// TwinCAT 3 PLC project Project
// ProgramVersion: 3.1.4023.0
// libraries:
//   Tc2_EtherCAT, * (Beckhoff Automation GmbH)
//   Tc2_Standard, * (Beckhoff Automation GmbH)
//   Tc2_System, * (Beckhoff Automation GmbH)
//   Tc2_Utilities, * (Beckhoff Automation GmbH)
//   Tc3_Module, * (Beckhoff Automation GmbH)
// project tree:
//   DUTs/ EtherCATDiagnosisState.TcDUT, SlaveInfo.TcDUT
//   GVLs/ GVL.TcGVL
//   / PlcTask.TcTTO
//   POUs/EtherCAT Monitoring/ FB_Diag_ECAT_Module.TcPOU, FB_EtherCATInit.TcPOU, FB_ReadSlavesEherCAT.TcPOU, SIC_Diagnosis_Modules.TcPOU
//   POUs/ MAIN.TcPOU
// real-time tasks:
//   TASK PlcTask: cycle T#1ms, priority 20, ADS port 350
// I/O:
//   DEVICE Device 1 (EtherCAT), AmsNetId 192.168.212.233.2.1
//     SyncCRIO (NI 9145) [NI 9145]
//     AZ5 (TW.LSST.AZIMUTH) [TW.LSST.AZIMUTH]
//     AZ6 (TW.LSST.AZIMUTH) [TW.LSST.AZIMUTH]
//     AZ7 (TW.LSST.AZIMUTH) [TW.LSST.AZIMUTH]
//     AZ8 (TW.LSST.AZIMUTH) [TW.LSST.AZIMUTH]
//     AZ_HS (LSST.HS.board) [LSST.HS.board]
//     AZ16 (TW.LSST.AZIMUTH) [TW.LSST.AZIMUTH]
//     AZ15 (TW.LSST.AZIMUTH) [TW.LSST.AZIMUTH]
//     AZ14 (TW.LSST.AZIMUTH) [TW.LSST.AZIMUTH]
//     AZ13 (TW.LSST.AZIMUTH) [TW.LSST.AZIMUTH]
//     EL51 (TW.LSST.ALTITUDE) [TW.LSST.ALTITUDE]
//     EL52 (TW.LSST.ALTITUDE) [TW.LSST.ALTITUDE]
//     EL41 (TW.LSST.ALTITUDE) [TW.LSST.ALTITUDE]
//     EL42 (TW.LSST.ALTITUDE) [TW.LSST.ALTITUDE]
//     EL_XNeg_HS (LSST.HS.board) [LSST.HS.board]
//     EL61 (TW.LSST.ALTITUDE) [TW.LSST.ALTITUDE]
//     EL62 (TW.LSST.ALTITUDE) [TW.LSST.ALTITUDE]
//     AZ9 (TW.LSST.AZIMUTH) [TW.LSST.AZIMUTH]
//     AZ10 (TW.LSST.AZIMUTH) [TW.LSST.AZIMUTH]
//     AZ11 (TW.LSST.AZIMUTH) [TW.LSST.AZIMUTH]
//     AZ12 (TW.LSST.AZIMUTH) [TW.LSST.AZIMUTH]
//     AZ4 (TW.LSST.AZIMUTH) [TW.LSST.AZIMUTH]
//     AZ3 (TW.LSST.AZIMUTH) [TW.LSST.AZIMUTH]
//     AZ2 (TW.LSST.AZIMUTH) [TW.LSST.AZIMUTH]
//     AZ1 (TW.LSST.AZIMUTH) [TW.LSST.AZIMUTH] (disabled)
//     EL21 (TW.LSST.ALTITUDE) [TW.LSST.ALTITUDE]
//     EL22 (TW.LSST.ALTITUDE) [TW.LSST.ALTITUDE]
//     EL11 (TW.LSST.ALTITUDE) [TW.LSST.ALTITUDE]
//     EL12 (TW.LSST.ALTITUDE) [TW.LSST.ALTITUDE]
//     EL_XPos_HS (LSST.HS.board) [LSST.HS.board]
//     EL31 (TW.LSST.ALTITUDE) [TW.LSST.ALTITUDE]
//     EL32 (TW.LSST.ALTITUDE) [TW.LSST.ALTITUDE]
// variable links:
//   Project/Project Instance <-> Device 1 (EtherCAT)/AZ5 (TW.LSST.AZIMUTH)
//     PlcTask Inputs/MAIN.StatusWordDrive2 <-> Inputs/Status word

CONFIGURATION Project
    RESOURCE PLC ON TwinCAT3
        TASK PlcTask(INTERVAL := T#1ms, PRIORITY := 20);
        PROGRAM MAIN WITH PlcTask : MAIN;
    END_RESOURCE
END_CONFIGURATION

// ---- DUTs/EtherCATDiagnosisState.TcDUT
{attribute 'qualified_only'}
{attribute 'strict'}
TYPE EtherCATDiagnosisState :
(
	Init								:= 0,
	GetPLCAdress						:= 1,
	GetSlavesAddresses 					:= 2,
	GetSlavesConfiguration 				:= 3,
	ReadSlavesIdentity					:= 4,
	
	ReadSlaveCyclicData					:= 10,
	
	ProcessSlavesCyclicData				:= 100
);
END_TYPE

// ---- DUTs/SlaveInfo.TcDUT
TYPE SlaveInfo :
STRUCT
	Address 						: WORD;
	Name 							: STRING[31];
	ConfiguredVendorID				: UDINT;
	ConfiguredProductCode 			: UDINT;
	ConfiguredRevisionNo 			: UDINT;
	ConfiguredSerialNo				: UDINT;
	ReadVendorID					: UDINT;
	ReadProductCode 				: UDINT;
	ReadRevisionNo 					: UDINT;
	ReadSerialNo					: UDINT;
	CRCerrorCounter					: DWORD;
	stCrcError						: ST_EcCrcErrorEx;
	StateChanges					: UDINT;
	StateChangesTimes				: ARRAY [0..255] OF TIMESTRUCT;
	StateChangesIndex				: UINT;
	AbnormalStateChanges			: UDINT;
	AbnormalStateChangesTimes		: ARRAY [0..255] OF TIMESTRUCT;
	AbnormalStateChangesIndex		: UINT;
	
	
END_STRUCT
END_TYPE

// ---- GVLs/GVL.TcGVL

VAR_GLOBAL
	PLCEtherCatAddress : T_AmsNetId;
END_VAR

// ---- POUs/MAIN.TcPOU
PROGRAM MAIN
VAR
	MyVar AT%I*:UDINT;
	StatusWordDrive2 AT%I*:UINT;
	
	
	b_PLCInitialization			: BOOL;
	b_EtherCATMasterErrorRun	: BOOL;
	
	//fbEtherCatInit 			: FB_EtherCATInit;
	
	
	
	fbGetLocalAmsNetId		: FB_GetLocalAmsNetId;
	sPlcNetId				: T_AmsNetId := '192.168.212.233.1.1';
	sEcatMaterNetId       	: T_AmsNetId := '192.168.212.233.2.1';
//	fbGetEcMasterState 		: FB_EcGetMasterState;
	 fbGetAllEcSlaveStates 	: FB_EcGetAllSlaveStates;
	 
    bExecute            : BOOL := TRUE;
    devStates           : ARRAY[0..EC_MAX_SLAVES] OF ST_EcSlaveState;
    nSlaves             : UINT := 0;
    bError              : BOOL;
    nErrId              : UDINT;
	
	bFirstCall 					: BOOL := TRUE;
	fbGetAllEcSlaveAddr 		: FB_EcGetAllSlaveAddr;
	slaveAddresses    			: ARRAY[0..EC_MAX_SLAVES] OF UINT;    
    bErrorSlaveAddr           	: BOOL;
  
	
	i : UINT;
	
	fbGetSlaveIdentity : FB_EcGetSlaveIdentity;  
    identity           : ARRAY [0..EC_MAX_SLAVES] OF ST_EcSlaveIdentity;
	
	fbEcGetConfSlaves : FB_EcGetConfSlaves;
	ArrEcConfSlaveInfo : ARRAY[0..EC_MAX_SLAVES] OF ST_EcSlaveConfigData; 
	
	
	fbEcGetAllSlavesStateChanges 	: FB_EcGetAllSlavePresentStateChanges;
	ArrSlaveStateChangeBuff	  		:  ARRAY [0..EC_MAX_SLAVES] OF UDINT;
	
	fbEcGetAllSlavesCrcErrors			: FB_EcGetAllSlaveCrcErrors;
	ArrSlavesCrcErrorCounterBuff	: ARRAY [0..EC_MAX_SLAVES] OF DWORD;
	
	fbEcGetSlaveCrcError		: FB_EcGetSlaveCrcError;
	
	fbEcGetAllSlaveAbnormalStateChanges	: FB_EcGetAllSlaveAbnormalStateChanges;
	ArrSlavesAbnormalStateChanges		:  ARRAY [0..EC_MAX_SLAVES] OF UDINT; 
    
	fbGetTime : NT_GetTime;
	
   bBusy : BOOL;
   
   
   arrSlaveData : ARRAY [0..EC_MAX_SLAVES] OF SlaveInfo;

	
	lastStateChangeValue: UDINT;
	
	eDiagnosisState : EtherCATDiagnosisState := EtherCATDiagnosisState.Init;
	
END_VAR

VAR CONSTANT
	EC_MAX_SLAVES : UINT :=255;
END_VAR


CASE eDiagnosisState OF
	//Init the diagnosis
	EtherCATDiagnosisState.Init:
		bExecute := TRUE;
		eDiagnosisState := EtherCATDiagnosisState.GetPLCAdress;
		FOR i:= 0 TO EC_MAX_SLAVES DO
			arrSlaveData[i].StateChangesIndex 			:= 0;
			arrSlaveData[i].AbnormalStateChangesIndex 	:= 0;
		END_FOR
 				
	//Get PLC address
	EtherCATDiagnosisState.GetPLCAdress:
		fbGetLocalAmsNetId(bExecute:= bExecute);
		bBusy := fbGetLocalAmsNetId.bBusy;
		bError := fbGetLocalAmsNetId.bError;
		IF NOT bBusy AND NOT bError AND bExecute THEN
			sPlcNetId := fbGetLocalAmsNetId.AddrString;
			eDiagnosisState := EtherCATDiagnosisState.GetSlavesAddresses;		
		END_IF
		
		IF bError THEN
			bExecute := FALSE;
		ELSE
			bExecute := TRUE;
		END_IF
		
	//Get EtherCAT slaves addresses
	EtherCATDiagnosisState.GetSlavesAddresses:
		fbGetAllEcSlaveAddr(sNetId:= sEcatMaterNetId,pAddrBuf := ADR(slaveAddresses), cbBufLen:= SIZEOF(slaveAddresses), bExecute:=bExecute);
		bBusy := fbGetAllEcSlaveAddr.bBusy;
		bError := fbGetAllEcSlaveAddr.bError;
		IF NOT bBusy AND NOT bError AND bExecute THEN
			nSlaves := fbGetAllEcSlaveAddr.nSlaves;
			FOR i:= 0 TO nSlaves-1 DO
				arrSlaveData[i].Address	:= slaveAddresses[i];
			END_FOR
			eDiagnosisState := EtherCATDiagnosisState.GetSlavesConfiguration;		
		END_IF
		
		IF bError THEN
			bExecute := FALSE;
		ELSE
			bExecute := TRUE;
		END_IF
		
	//Get salves configuration
	EtherCATDiagnosisState.GetSlavesConfiguration:
		fbEcGetConfSlaves(sNetId:= sEcatMaterNetId, pArrEcConfSlaveInfo:= ADR(ArrEcConfSlaveInfo), cbBufLen:= SIZEOF(ArrEcConfSlaveInfo), bExecute:= bExecute);
		bBusy := fbEcGetConfSlaves.bBusy;
		bError := fbEcGetConfSlaves.bError;
		IF NOT bBusy AND NOT bError AND bExecute THEN			
			FOR i:= 0 TO nSlaves-1 DO
				arrSlaveData[i].ConfiguredProductCode	:= ArrEcConfSlaveInfo[i].stSlaveIdentity.productCode;
				arrSlaveData[i].ConfiguredRevisionNo	:= ArrEcConfSlaveInfo[i].stSlaveIdentity.revisionNo;
				arrSlaveData[i].ConfiguredSerialNo		:= ArrEcConfSlaveInfo[i].stSlaveIdentity.serialNo;
				arrSlaveData[i].ConfiguredVendorID		:= ArrEcConfSlaveInfo[i].stSlaveIdentity.vendorId;
				arrSlaveData[i].Name 					:= ArrEcConfSlaveInfo[i].sName;
				arrSlaveData[i].Address					:= ArrEcConfSlaveInfo[i].nAddr;
			END_FOR
			eDiagnosisState := EtherCATDiagnosisState.ReadSlavesIdentity;
			i := 0;		
		END_IF
		
		IF bError THEN
			bExecute := FALSE;
		ELSE
			bExecute := TRUE;
		END_IF
		
	//Read salves identity
	EtherCATDiagnosisState.ReadSlavesIdentity:
		
		fbGetSlaveIdentity(sNetId:= sEcatMaterNetId, nSlaveAddr:= arrSlaveData[i].Address, bExecute:=bExecute);
		bBusy := fbEcGetConfSlaves.bBusy;
		bError := fbEcGetConfSlaves.bError;
		IF NOT bBusy AND NOT bError AND bExecute THEN			
			arrSlaveData[i].ReadProductCode 		:= fbGetSlaveIdentity.identity.productCode;
			arrSlaveData[i].ReadRevisionNo 			:= fbGetSlaveIdentity.identity.revisionNo;
			arrSlaveData[i].ReadSerialNo 			:= fbGetSlaveIdentity.identity.serialNo;
			arrSlaveData[i].ReadVendorID 			:= fbGetSlaveIdentity.identity.vendorId;
			i := i+1;						
		END_IF
			
		IF bError THEN
			bExecute := FALSE;
		ELSE
			IF bBusy THEN
				bExecute := TRUE;
			ELSE
				bExecute := NOT bExecute;
			END_IF
		END_IF
		
		IF i>=nSlaves THEN
			eDiagnosisState := EtherCATDiagnosisState.ReadSlaveCyclicData;
			bExecute 		:= TRUE;
		END_IF
		
		
	//read slaves cyclic data
	EtherCATDiagnosisState.ReadSlaveCyclicData:
		bError := FALSE;
		bBusy  := FALSE;
		fbGetAllEcSlaveStates(sNetId:= sEcatMaterNetId, pStateBuf := ADR(devStates), cbBufLen:=SIZEOF(devStates), bExecute:=bExecute);
		bError := bError OR fbGetAllEcSlaveStates.bError;
		bBusy := bBusy OR fbGetAllEcSlaveStates.bBusy;
		
		fbEcGetAllSlavesCrcErrors(sNetId:= sEcatMaterNetId, pCrcErrorBuf:= ADR(ArrSlavesCrcErrorCounterBuff), cbBufLen:= SIZEOF(ArrSlavesCrcErrorCounterBuff), bExecute:= bExecute);
		bError := bError OR fbEcGetAllSlavesCrcErrors.bError;
		bBusy := bBusy OR fbEcGetAllSlavesCrcErrors.bBusy;
		
		fbEcGetAllSlavesStateChanges(sNetId:= sEcatMaterNetId, pAddrBuf:= ADR(ArrSlaveStateChangeBuff), cbBufLen:= SIZEOF(ArrSlaveStateChangeBuff), bExecute:= bExecute);
		bError := bError OR fbEcGetAllSlavesStateChanges.bError;
		bBusy := bBusy OR fbEcGetAllSlavesStateChanges.bBusy;
		
		fbEcGetAllSlaveAbnormalStateChanges(sNetId:= sEcatMaterNetId, pAddrBuf:= ADR(ArrSlavesAbnormalStateChanges), cbBufLen:= SIZEOF(ArrSlavesAbnormalStateChanges), bExecute:= bExecute);
		bError := bError OR fbEcGetAllSlaveAbnormalStateChanges.bError;
		bBusy := bBusy OR fbEcGetAllSlaveAbnormalStateChanges.bBusy;

		fbGetTime(NETID:=sPlcNetId, START:=bExecute);
		
		IF NOT bBusy AND NOT bError AND bExecute THEN
			eDiagnosisState := EtherCATDiagnosisState.ProcessSlavesCyclicData;
		END_IF
		
		IF bError THEN
			bExecute := FALSE;
		ELSE
			bExecute := TRUE;
		END_IF
		
		//Process salves cyclic data
		EtherCATDiagnosisState.ProcessSlavesCyclicData:
			FOR i:=0 TO nSlaves-1 DO
				lastStateChangeValue 			:= arrSlaveData[i].StateChanges;
				arrSlaveData[i].StateChanges 	:= ArrSlaveStateChangeBuff[i];
				IF arrSlaveData[i].StateChanges <> lastStateChangeValue THEN					
					arrSlaveData[i].StateChangesTimes[arrSlaveData[i].StateChangesIndex] := fbGetTime.TIMESTR; 
					arrSlaveData[i].StateChangesIndex := arrSlaveData[i].StateChangesIndex + 1;					
				END_IF		
                lastStateChangeValue                    := arrSlaveData[i].AbnormalStateChanges;
                arrSlaveData[i].AbnormalStateChanges 	:= ArrSlavesAbnormalStateChanges[i];
                IF arrSlaveData[i].AbnormalStateChanges <> lastStateChangeValue THEN
                    arrSlaveData[i].AbnormalStateChangesTimes[arrSlaveData[i].AbnormalStateChangesIndex] := fbGetTime.TIMESTR; 
                    arrSlaveData[i].AbnormalStateChangesIndex := arrSlaveData[i].AbnormalStateChangesIndex + 1;
                END_IF
                arrSlaveData[i].CRCerrorCounter			:= ArrSlavesCrcErrorCounterBuff[i];
            END_FOR
            bExecute := FALSE;
            eDiagnosisState := EtherCATDiagnosisState.ReadSlaveCyclicData;
		ELSE
			bExecute := FALSE;
		
END_CASE

END_PROGRAM

// ---- POUs/EtherCAT Monitoring/FB_Diag_ECAT_Module.TcPOU
FUNCTION_BLOCK FB_Diag_ECAT_Module
VAR_INPUT
	bWCounter	:BIT;
	wState		:WORD;
	TimeError	:TIME;
END_VAR
VAR_OUTPUT
	bError		:BOOL;
END_VAR
VAR
	iStOP		: INT;
	wStateWord	: WORD;
	TONErroR	: TON;
END_VAR

wStateWord := wstate AND 16#000F;

TONError(IN:= (bWcounter = 1 OR wStateWord <> 8),PT:=TimeError);
bError:=TONError.Q;

END_FUNCTION_BLOCK

// ---- POUs/EtherCAT Monitoring/FB_EtherCATInit.TcPOU
FUNCTION_BLOCK FB_EtherCATInit
VAR_INPUT
	iADSAmsNetId : ARRAY[0..5] OF BYTE;
END_VAR
VAR_OUTPUT	
	oPLCInicialization		: BOOL; 		// PLC Initiliation OK
	oECatMasterError 		: BOOL;		// MasterECat Error
	oSlavesECatError 		: BOOL;		// Slaves State Error NOT OP
	oErrorPLCInicialization : INT; // Error ID
	oDeviceECATNoInit		:ST_InfoEtherCATSlaves; // EtherCAT slave Not Init
END_VAR

VAR_IN_OUT
	ioFirstCyclePlc : BOOL;
END_VAR
	
VAR
	arSlavesData : ARRAY[0..nNumberSlaves] OF ST_InfoEtherCATSlaves;	(* Struct to save data read*)
	bExecute1 : BOOL; 										(* Function Execute Signal*)
	FBReadSlaves: FB_ReadSlavesEherCAT; 					(* Function to read EherCAT Slaves*)
		
	InitNo				:INT:=0;		// 0 para realizar la inicialización Ó 5 para no chequear hw
	bExecute			:BOOL;
	bUsersLoaded		:BOOL:=FALSE;
	i					:INT;
	
	FBEcGetMasterState:FB_EcGetMasterState;
	FBEcSetMasterState:FB_EcSetMasterState;

END_VAR

VAR CONSTANT
	nNumberSlaves : INT := 14;
END_VAR

VAR PERSISTENT
	(* READ ONLY: TRUE when all PLC variables are updated with database info *)
	bDataReady_out : BOOL := FALSE;
	(* READ ONLY: 0 when no errors happened and >0 otherwise *)
	nDataErrors_out : UINT := 0;
END_VAR

// PLC Inicialization
CASE InitNo OF
	0:	// Get ADSAmsNetId
		PLCEtherCatAddress:=F_CreateAmsNetId(nIds:=iADSAmsNetId);
		IF PLCEtherCatAddress <> '' 
		THEN 
			InitNo:=1;	//	Next Step
		END_IF;
		
	1:	//Get Status 
		bExecute:= NOT bExecute;
		FBEcGetMasterState(
			sNetId:=PLCEtherCatAddress,
			bExecute:=bExecute,
			tTimeout:=t#10s,
			bBusy=> ,
			bError=> ,
			nErrId=> ,
			state=> );

		IF FBEcGetMasterState.state=8 
		THEN 
			InitNo:=3;	//	Next Step
			FBEcGetMasterState(bExecute:=FALSE );
		ELSIF FBEcGetMasterState.state=1 
		THEN 
			InitNo:=2;	//	Set Status
			FBEcGetMasterState(bExecute:=FALSE );
		END_IF
		
		IF FBEcGetMasterState.bError 
		THEN
			InitNo:= 7;					// Initialization_Error
			oECatMasterError:=TRUE;	// EtherCAT Master Error
		END_IF

	2:	// Set Status 8 if does not work, NOT OP
		FBEcSetMasterState(
			sNetId:=PLCEtherCatAddress,
			bExecute:= TRUE,
			tTimeout:= t#10s,
			reqState:=8 ,
			bBusy=> ,
			bError=> ,
			nErrId=> ,
			currState=> );

		bExecute:= NOT bExecute;

		FBEcGetMasterState(
			sNetId:=PLCEtherCatAddress,
			bExecute:=bExecute,
			tTimeout:=t#10s,
			bBusy=> ,
			bError=> ,
			nErrId=> , 
			state=> );
		
		IF FBEcGetMasterState.bError OR FBEcSetMasterState.bError 
		THEN
			InitNo:=7;						// Initialization_Error
			oECatMasterError := TRUE;		// EtherCAT Master Error
			oErrorPLCInicialization := 1;
		END_IF; 
		
		IF FBEcGetMasterState.state=8 
		THEN 
			InitNo:=3;	//	Next Step
		END_IF

		InitNo:=3;	//	Next Step
		
	3:	// Get Status of EtherCAT Slaves
		FBReadSlaves(sNetID:=PLCEtherCatAddress ,
					 pArray:= ADR(arSlavesData), 
					 nSizeStruct:=SIZEOF(arSlavesData),
					 bExecute:= ioFirstCyclePlc) ;
		IF NOT FBReadSlaves.bBusy 
		THEN
			IF FBReadSlaves.bDone
			THEN
				InitNo:=4;	//	Next Step
			ELSIF FBReadSlaves.bError 
			THEN
				InitNo:=7; // Not initialization
				InitNo:=4;
			END_IF
		END_IF
			
	4:	// Check the Status of Slaves		
		FOR i:=0 TO nNumberSlaves-1 DO
			IF arSlavesData[i].enState <> Operational_State AND NOT oSlavesECatError
			THEN
				oSlavesECatError := TRUE;
				oDeviceECATNoInit	:=	arSlavesData[i];	//Save the Slave with Error
			END_IF
		END_FOR
		IF oSlavesECatError
		THEN			
			InitNo:=7;
			oErrorPLCInicialization := 3;		//Error in Parameters Load
		ELSE
			InitNo:=6;	//	No Error
		END_IF	

	6:
		ioFirstCyclePlc := FALSE;  		// End Initialization
		oPLCInicialization:=TRUE; 		// PLC Initiliation OK
		oECatMasterError:=FALSE;		// MasterECat Error
		oSlavesECatError:=FALSE;		// Slaves State Error NOT OP
		
	7:
		ioFirstCyclePlc := FALSE;		// End Initialization
		oPLCInicialization:=FALSE;		// PLC Initiliation  NO OK
		
END_CASE

END_FUNCTION_BLOCK

// ---- POUs/EtherCAT Monitoring/FB_ReadSlavesEherCAT.TcPOU
FUNCTION_BLOCK FB_ReadSlavesEherCAT
VAR_INPUT
	bExecute:BOOL; (*Execute*)
	sNetID: T_AmsNetId; (*AMS Address of EtherCAT Master*)
	pArray: POINTER TO ARRAY[0..iNumberSlaves] OF st_InfoEtherCATSlaves; (*(14 number of slaves)A pointer to the memory address where the data stored start*)
	nSizeStruct: UDINT; (*Bytes number to modify in the reading*)
END_VAR
VAR_OUTPUT
	bError: BOOL:= FALSE; 	(* Error Reading the slaves*)
	bDone : BOOL := FALSE;	(* Finished reading the slaves*)
	bBusy : BOOL := FALSE; 	(* Function busy*)
	nErrorID: UINT:=0; 		(* State where the error occurs *)
	nEtherCATSlaves : UINT := 0; (*number of EtherCAT Slaves*)
END_VAR
VAR
	stLocalInfoEtherCATSlave : st_InfoEtherCATSlaves; (*Current data of slave*)
	nEstado: UINT:=0; (*Current value of State Machine*)
	nIndex: UINT (*Number of slaves reading at the moment*);
	RisingEdge:R_TRIG; 
	nSlaves: UINT :=0; (*Number of slaves EtherCAT detected*)
	fbGetSlaveCount : FB_EcGetSlaveCount; (*Reading slave Function*)
	tTimeout	: TIME := DEFAULT_ADS_TIMEOUT; (*Maximum time to execute the reader function of slaves*)
	(*Variables to read the NAMES*)
	stLocalInfo: ST_EcSlaveConfigData; (*Aux variable to save the NAME and ADDRESS of the slaves*)
	fbAdsRead: ADSREAD; (*Reading function to get slaves data*)
	nIdxOffs: UDINT; (*Offset to indicate wich slave to get data*)
	(*Constant to calculate the offset*)
	nSDO_IDX_SBP_SLAVECONFIGDATASTART : DWORD := 16#00_00_80_00;
	nADSIOFFS_ECAT_COE_COMPLETEACCESS : DWORD := 16#00_00_01_00;
	(*Variable to CRC*)
	fbGetSlaveCrcError : FB_EcGetSlaveCrcError; (*CRC Reader function of a slave*)
	(*Variable to read States of slaves*)
	fbGetSlaveState: FB_EcGetSlaveState;  (*Reader function to get de operation state and connection of a slaves*)
END_VAR

VAR CONSTANT
	iNumberSlaves : INT := 19;
END_VAR

CASE nEstado OF
	0:      
		RisingEdge( CLK:= bExecute );
		(*Initialization of variables *)
		IF RisingEdge.Q 
		THEN
			bBusy 		:= TRUE;
			bError 		:= FALSE;
			bDone		:= FALSE;
			nErrorId 	:= 0;
			nSlaves		:= 0;
			MEMSET( pArray, 0, nSizeStruct ); (*Delete old information of EtherCAT Slaves*)
			nEstado		:= 10;
			nIndex 		:=	1;
		END_IF

	10:    (*Get the counter of slaves connected*)
		fbGetSlaveCount(sNetId:= sNetId, 
						bExecute:=TRUE);
		nSlaves:=fbGetSlaveCount.nSlaves;

		(*Reading finished and all is OK *)
		IF NOT fbGetSlaveCount.bBusy AND NOT fbGetSlaveCount.bError 
		THEN
			(*Check that any slave is connected, if not finish*)
			IF nSlaves = 0 
			THEN
				nEstado:=11;
				nIndex :=0; (* Set this value to out in State 60*)
				fbGetSlaveCount(sNetId:= sNetId, bExecute:=FALSE);
			(*Any slave connected*)
			ELSE
				nEstado:=20;
				fbGetSlaveCount(sNetId:= sNetId, 
								bExecute:=FALSE);
			END_IF
		END_IF

		(*GetSlave Error -- go to State 50*)
		IF fbGetSlaveCount.bError 
		THEN
			fbGetSlaveCount(sNetId:= sNetId, bExecute:=FALSE);
			bError		:=TRUE;
			bBusy		:=FALSE;
			nErrorID	:=nEstado;
			bDone		:=FALSE;
			nEstado		:=0;
		END_IF

	11:	(*No EtherCAT slave detected*)
		bError		:= TRUE;
		bBusy		:= FALSE;
		nErrorID	:= nEstado;
		bDone		:= FALSE;
		nEstado		:= 0;

	20:    (*Name and Address of slaves*)
		nIdxOffs := SHL(nSDO_IDX_SBP_SLAVECONFIGDATASTART+(nIndex-1),16) OR nADSIOFFS_ECAT_COE_COMPLETEACCESS; (*Calculate the offset to indicate the slave to ask for information*)
		fbAdsRead(NETID:= sNetId,PORT:= EC_AMSPORT_MASTER,IDXGRP:= EC_ADS_IGRP_CANOPEN_SDO,IDXOFFS:= nIdxOffs,LEN:= SIZEOF(stLocalInfo),DESTADDR:= ADR(stLocalInfo),	READ:= TRUE,TMOUT:= tTimeout);

		(*Finish the reading and all is OK, go to Next State *)
		IF NOT fbAdsRead.Busy AND NOT fbAdsRead.Err 
		THEN
			stLocalInfoEtherCATSlave.nAddress:=stLocalInfo.nAddr;
			stLocalInfoEtherCATSlave.sName:=stLocalInfo.sName;
			nEstado:=30;
			fbAdsRead( READ := FALSE );
		END_IF

		(*Any error in Reading, go to State 50*)
		IF fbAdsRead.Err 
		THEN
			stLocalInfoEtherCATSlave.nErrorLectura := nEstado;
			nEstado:=50;
			fbAdsRead( READ := FALSE );
		END_IF

	30:    (*Reading CRCs of slaves*)
		fbGetSlaveCrcError(sNetId:= sNetId, 
						   nSlaveAddr:= stLocalInfo.nAddr, 
						   bExecute:=TRUE);

		(*Finish the reading and all is OK, go to Next State *)
		IF NOT fbGetSlaveCrcError.bBusy AND NOT fbGetSlaveCrcError.bError 
		THEN
			stLocalInfoEtherCATSlave.dwCRC:=(fbGetSlaveCrcError.crcError.portA+fbGetSlaveCrcError.crcError.portB+fbGetSlaveCrcError.crcError.portC); (*El CRC que devuelve es la suma del CRC de cada puerto*)
			nEstado:=40;
			fbGetSlaveCrcError(bExecute:=FALSE);
		END_IF

		(*Any error in REading, go to State 50*)
		IF fbGetSlaveCrcError.bError 
		THEN
			stLocalInfoEtherCATSlave.nErrorLectura := nEstado;
			nEstado:=50;
			fbGetSlaveCrcError(bExecute:=FALSE);
		END_IF

	40:   (*Reading state of the slaves*)
		fbGetSlaveState(sNetId:= sNetId, nSlaveAddr:= stLocalInfo.nAddr, bExecute:=TRUE);

		(*Finish the reading and all is OK, go to Next State *)
		IF NOT fbGetSlaveState.bBusy AND NOT fbGetSlaveState.bError 
		THEN
			stLocalInfoEtherCATSlave.nLink:=fbGetSlaveState.state.linkState;
			stLocalInfoEtherCATSlave.enState:=fbGetSlaveState.state.deviceState;
			stLocalInfoEtherCATSlave.bErrorLectura:=FALSE; (*to be in this point mean all data read correctly*)
			stLocalInfoEtherCATSlave.nErrorLectura := 0;
			nEstado:=60;
			fbGetSlaveState(bExecute:=FALSE);
		END_IF

		(*Any error in REading, go to State 50*)
		IF fbGetSlaveState.bError 
		THEN
			stLocalInfoEtherCATSlave.nErrorLectura := nEstado;
			nEstado:=50;
			fbGetSlaveState(bExecute:=FALSE);
		END_IF

	50:    (*Any Error in Reading*)
		stLocalInfoEtherCATSlave.bErrorLectura:=TRUE;
		nEstado :=60;

	60:   (*Write in out memory*)
		(*Any slave was detedted*)
		IF nSlaves > 0 
		THEN
			MEMCPY(pArray + UINT_TO_UDINT(nIndex-1)*SIZEOF(stLocalInfoEtherCATSlave), ADR(stLocalInfoEtherCATSlave), SIZEOF(stLocalInfoEtherCATSlave));
		END_IF
		(*All slaves indicated are read, go to initial state*)
		IF nIndex = nSizeStruct/SIZEOF(stLocalInfoEtherCATSlave) OR nIndex = nSlaves 
		THEN
			nEstado := 0;
			bDone := TRUE;
			bBusy := FALSE;
			bError := FALSE;
			nEtherCATSlaves := nSlaves;
		(*More slaves to read, go to State 20 to read the next*)
		ELSE
			nEstado := 20;
			nIndex := nIndex + 1;
		END_IF
END_CASE

END_FUNCTION_BLOCK

// ---- POUs/EtherCAT Monitoring/SIC_Diagnosis_Modules.TcPOU
PROGRAM SIC_Diagnosis_Modules
VAR
	(**********************************************************)
	(* 					EtherCAT Master						  *)
	(**********************************************************)
//	{attribute 'TcLinkTo' := 'TIID^EtherCAT_Master (EtherCAT)^InfoData^AmsNetId'}
//	ADSAmsNetId	AT %I* : ARRAY[0..5] OF BYTE;
	
	

	// EtheCAT Diagnosis
	bExe							: BOOL;
	FBEcGetMasterState				: FB_EcGetMasterState;
	FB_EcMasterFrameStatistic 		: FB_EcMasterFrameStatistic;
	bExecute						: BOOL;
	
	// 1. Bus Coupler 1 
	FBDiagnosis_201KF11		:	FB_Diag_ECAT_Module();
	FBDiagnosis_201KF21		:	FB_Diag_ECAT_Module();
	FBDiagnosis_201KF22		:	FB_Diag_ECAT_Module();
	FBDiagnosis_201KF23		:	FB_Diag_ECAT_Module();
	FBDiagnosis_201KF31		:	FB_Diag_ECAT_Module();
	FBDiagnosis_201KF41		:	FB_Diag_ECAT_Module();
	FBDiagnosis_201KF42		:	FB_Diag_ECAT_Module();
	FBDiagnosis_201KF43		:	FB_Diag_ECAT_Module();
	FBDiagnosis_201KF51		:	FB_Diag_ECAT_Module();
	FBDiagnosis_201KF61		:	FB_Diag_ECAT_Module();
	FBDiagnosis_201KF62		:	FB_Diag_ECAT_Module();
	FBDiagnosis_201KF71		:	FB_Diag_ECAT_Module();
	FBDiagnosis_201KF72		:	FB_Diag_ECAT_Module();
	FBDiagnosis_201KF81		:	FB_Diag_ECAT_Module();
	FBDiagnosis_201KF91		:	FB_Diag_ECAT_Module();	
	FBDiagnosis_101TB1		:	FB_Diag_ECAT_Module();
	FBDiagnosis_101TB2		:	FB_Diag_ECAT_Module();
	FBDiagnosis_101TB3		:	FB_Diag_ECAT_Module();
	FBDiagnosis_101TB4		:	FB_Diag_ECAT_Module();	
	
	// Bus Coupler 1
	// -201KF11
	{attribute 'TcLinkTo' := 'TIID^EtherCAT_Master (EtherCAT)^-201KF11 (EK1100)^InfoData^State'}	
	ui201BC1State	AT	%I*:	UINT;	// State 
	
	// -201KF21
	{attribute 'TcLinkTo' := 'TIID^EtherCAT_Master (EtherCAT)^-201KF11 (EK1100)^-201KF21 (EL1008)^WcState^WcState'}
	b201DI1Wc			AT	%I*:	BOOL;	// Working Counter
	{attribute 'TcLinkTo' := 'TIID^EtherCAT_Master (EtherCAT)^-201KF11 (EK1100)^-201KF21 (EL1008)^InfoData^State'}
	ui201DI1State		AT	%I*:	UINT;	// State
	
	// -201KF22
	{attribute 'TcLinkTo' := 'TIID^EtherCAT_Master (EtherCAT)^-201KF11 (EK1100)^-201KF22 (EL1008)^WcState^WcState'}
	b201DI2Wc			AT	%I*:	BOOL;	// Working Counter
	{attribute 'TcLinkTo' := 'TIID^EtherCAT_Master (EtherCAT)^-201KF11 (EK1100)^-201KF22 (EL1008)^InfoData^State'}
	ui201DI2State		AT	%I*:	UINT;	// State
	
	// -201KF23
	{attribute 'TcLinkTo' := 'TIID^EtherCAT_Master (EtherCAT)^-201KF11 (EK1100)^-201KF23 (EL1008)^WcState^WcState'}
	b201DI3Wc			AT	%I*:	BOOL;	// Working Counter
	{attribute 'TcLinkTo' := 'TIID^EtherCAT_Master (EtherCAT)^-201KF11 (EK1100)^-201KF23 (EL1008)^InfoData^State'}
	ui201DI3State		AT	%I*:	UINT;	// State
	
	// -201KF31
	{attribute 'TcLinkTo' := 'TIID^EtherCAT_Master (EtherCAT)^-201KF11 (EK1100)^-201KF31 (EL3062)^WcState^WcState'}
	b201DAI1Wc			AT	%I*:	BOOL;	// Working Counter
	{attribute 'TcLinkTo' := 'TIID^EtherCAT_Master (EtherCAT)^-201KF11 (EK1100)^-201KF31 (EL3062)^InfoData^State'}
	ui201AI1State		AT	%I*:	UINT;	// State
	
	// -201KF41
	{attribute 'TcLinkTo' := 'TIID^EtherCAT_Master (EtherCAT)^-201KF11 (EK1100)^-201KF41 (EL1904)^WcState^WcStateIn'}
	b201SI2Wc			AT	%I*:	BOOL;	// Working Counter
	{attribute 'TcLinkTo' := 'TIID^EtherCAT_Master (EtherCAT)^-201KF11 (EK1100)^-201KF41 (EL1904)^InfoData^State'}
	ui201SI2State		AT	%I*:	UINT;	// State
	
	// -201KF42
	{attribute 'TcLinkTo' := 'TIID^EtherCAT_Master (EtherCAT)^-201KF11 (EK1100)^-201KF42 (EL1904)^WcState^WcStateIn'}
	b201SI3Wc			AT	%I*:	BOOL;	// Working Counter
	{attribute 'TcLinkTo' := 'TIID^EtherCAT_Master (EtherCAT)^-201KF11 (EK1100)^-201KF42 (EL1904)^InfoData^State'}
	ui201SI3State		AT	%I*:	UINT;	// State
	
	// -201KF43
	{attribute 'TcLinkTo' := 'TIID^EtherCAT_Master (EtherCAT)^-201KF11 (EK1100)^-201KF43 (EL1904)^WcState^WcStateIn'}
	b201SI4Wc			AT	%I*:	BOOL;	// Working Counter
	{attribute 'TcLinkTo' := 'TIID^EtherCAT_Master (EtherCAT)^-201KF11 (EK1100)^-201KF43 (EL1904)^InfoData^State'}
	ui201SI4State		AT	%I*:	UINT;	// State
	
	// -201KF51
	{attribute 'TcLinkTo' := 'TIID^EtherCAT_Master (EtherCAT)^-201KF11 (EK1100)^-201KF51 (EL6910)^WcState^WcStateIn'}
	b201SI1Wc			AT	%I*:	BOOL;	// Working Counter
	{attribute 'TcLinkTo' := 'TIID^EtherCAT_Master (EtherCAT)^-201KF11 (EK1100)^-201KF51 (EL6910)^InfoData^State'}
	ui201SI1State		AT	%I*:	UINT;	// State
	
	// -201KF61
	{attribute 'TcLinkTo' := 'TIID^EtherCAT_Master (EtherCAT)^-201KF11 (EK1100)^-201KF61 (EL2008-0015)^WcState^WcState'}
	b201DO1Wc			AT	%I*:	BOOL;	// Working Counter
	{attribute 'TcLinkTo' := 'TIID^EtherCAT_Master (EtherCAT)^-201KF11 (EK1100)^-201KF61 (EL2008-0015)^InfoData^State'}
	ui201DO1State		AT	%I*:	UINT;	// State
	
	// -201KF62
	{attribute 'TcLinkTo' := 'TIID^EtherCAT_Master (EtherCAT)^-201KF11 (EK1100)^-201KF62 (EL2068)^WcState^WcStateIn'}
	b201DO2Wc			AT	%I*:	BOOL;	// Working Counter
	{attribute 'TcLinkTo' := 'TIID^EtherCAT_Master (EtherCAT)^-201KF11 (EK1100)^-201KF62 (EL2068)^InfoData^State'}
	ui201DO2State		AT	%I*:	UINT;	// State
	
	// -201KF71
	{attribute 'TcLinkTo' := 'TIID^EtherCAT_Master (EtherCAT)^-201KF11 (EK1100)^-201KF71 (EL2904)^WcState^WcStateIn'}
	b201SO1Wc			AT	%I*:	BOOL;	// Working Counter
	{attribute 'TcLinkTo' := 'TIID^EtherCAT_Master (EtherCAT)^-201KF11 (EK1100)^-201KF71 (EL2904)^InfoData^State'}
	ui201SO1State		AT	%I*:	UINT;	// State
	
	// -201KF72
	{attribute 'TcLinkTo' := 'TIID^EtherCAT_Master (EtherCAT)^-201KF11 (EK1100)^-201KF72 (EL2904)^WcState^WcStateIn'}
	b201SO2Wc			AT	%I*:	BOOL;	// Working Counter
	{attribute 'TcLinkTo' := 'TIID^EtherCAT_Master (EtherCAT)^-201KF11 (EK1100)^-201KF72 (EL2904)^InfoData^State'}
	ui201SO2State		AT	%I*:	UINT;	// State	
	
	// -201KF81
	{attribute 'TcLinkTo' := 'TIID^EtherCAT_Master (EtherCAT)^-201KF11 (EK1100)^-201KF81 (EL9410)^WcState^WcState'}
	b201ST1Wc			AT	%I*:	BOOL;	// Working Counter
	{attribute 'TcLinkTo' := 'TIID^EtherCAT_Master (EtherCAT)^-201KF11 (EK1100)^-201KF81 (EL9410)^InfoData^State'}
	ui201ST1State		AT	%I*:	UINT;	// State
	
	// -201KF91
	{attribute 'TcLinkTo' := 'TIID^EtherCAT_Master (EtherCAT)^-201KF11 (EK1100)^-201KF91 (EL6631)^WcState^WcStateIn'}
	b201CO1Wc			AT	%I*:	BOOL;	// Working Counter
	{attribute 'TcLinkTo' := 'TIID^EtherCAT_Master (EtherCAT)^-201KF11 (EK1100)^-201KF91 (EL6631)^InfoData^State'}
	ui201CO1State		AT	%I*:	UINT;	// State
	
	// -101TB1
	{attribute 'TcLinkTo' := 'TIID^EtherCAT_Master (EtherCAT)^-101TB1 (AX5201-0000-0214)^InfoData^State'}
	ui101U1State		AT	%I*:	UINT;	// State
	
	// -101TB2
	{attribute 'TcLinkTo' := 'TIID^EtherCAT_Master (EtherCAT)^-101TB2 (AX5201-0000-0214)^InfoData^State'}
	ui101U2State		AT	%I*:	UINT;	// State
	
	// -101TB3
	{attribute 'TcLinkTo' := 'TIID^EtherCAT_Master (EtherCAT)^-101TB3 (AX5203-0000-0214)^InfoData^State'}
	ui101U3State		AT	%I*:	UINT;	// State
	
	// -101TB4
	{attribute 'TcLinkTo' := 'TIID^EtherCAT_Master (EtherCAT)^-101TB4 (AX5203-0000-0214)^InfoData^State'}
	ui101U4State		AT	%I*:	UINT;	// State
	
	

	
	

	
	
END_VAR

(*************** ETHERCAT DIAGNOSIS ************************************)
(* 1. EtherCAT Master State *)
bExe := NOT bExe;
FBEcGetMasterState(
			sNetId:=PLCEtherCatAddress,
			bExecute:=bExe,
			tTimeout:=t#10s,
			bBusy=> ,
			bError=> ,
			nErrId=> ,
			state=> );
			
b_EtherCATMasterErrorRun := b_PLCInitialization AND (FBEcGetMasterState.state <> 8);

(* State of the EtherCAT Frames *)
IF FBEcGetMasterState.state = 8 AND b_Pulse_1sec
THEN
	bExecute:= NOT bExecute;
	FB_EcMasterFrameStatistic(sNetId := PLCEtherCatAddress,
							  bExecute := bExecute);
END_IF
EtherCATMaster.udiLostFrames				:= FB_EcMasterFrameStatistic.nLostFrames;
EtherCATMaster.lrfFramesPerSecond			:= FB_EcMasterFrameStatistic.fFramesPerSecond;
EtherCATMaster.udinLostQueuedFrames			:= FB_EcMasterFrameStatistic.nLostQueuedFrames;
EtherCATMaster.lrfQueuedFramesPerSencond	:= FB_EcMasterFrameStatistic.fQueuedFramesPerSecond;

(*************** DIAGNOSIS OF ETHERCAT MODULES ********************)
(* -201 *)
FBDiagnosis_201KF11(bWCounter := FALSE,
				   wState := ui201BC1State,
				   TimeError :=Time100ms,
				   bError=> b_201BC1Error);
				   
FBDiagnosis_201KF21(bWCounter := FALSE,
				   wState := ui201BC1State,
				   TimeError :=Time100ms,
				   bError=> b_201DI1Error);
				   
FBDiagnosis_201KF22(bWCounter := FALSE,
				   wState := ui201DI2State,
				   TimeError :=Time100ms,
				   bError=> b_201DI2Error);
				   
FBDiagnosis_201KF23(bWCounter := FALSE,
				   wState := ui201DI3State,
				   TimeError :=Time100ms,				   
				   bError=> b_201DI3Error);
				   
FBDiagnosis_201KF31(bWCounter := FALSE,
				   wState := ui201AI1State,
				   TimeError :=Time100ms,
				   bError=> b_201AI1Error);

FBDiagnosis_201KF42(bWCounter := FALSE,
				   wState := ui201SI2State,
				   TimeError :=Time100ms,
				   bError=> b_201SI2Error);

FBDiagnosis_201KF43(bWCounter := FALSE,
				   wState := ui201SI3State,
				   TimeError :=Time100ms,
				   bError=> b_201SI3Error);

FBDiagnosis_201KF51(bWCounter := FALSE,
				   wState := ui201SI4State,
				   TimeError :=Time100ms,
				   bError=> b_201SI4Error);

FBDiagnosis_201KF41(bWCounter := FALSE,
				   wState := ui201SI1State,
				   TimeError :=Time100ms,
				   bError=> b_201SI1Error);

FBDiagnosis_201KF61(bWCounter := FALSE,
				   wState := ui201DO1State,
				   TimeError :=Time100ms,
				   bError=> b_201DO1Error);

FBDiagnosis_201KF62(bWCounter := FALSE,
				   wState := ui201DO2State,
				   TimeError :=Time100ms,
				   bError=> b_201DO2Error);

FBDiagnosis_201KF71(bWCounter := FALSE,
				   wState := ui201SO1State,
				   TimeError :=Time100ms,
				   bError=> b_201SO1Error);
				   
FBDiagnosis_201KF72(bWCounter := FALSE,
				   wState := ui201SO2State,
				   TimeError :=Time100ms,
				   bError=> b_201SO2Error);

FBDiagnosis_201KF81(bWCounter := FALSE,
				   wState := ui201ST1State,
				   TimeError :=Time100ms,
				   bError=> b_201ST1Error);

FBDiagnosis_201KF91(bWCounter := FALSE,
				   wState := ui201CO1State,
				   TimeError :=Time100ms,
				   bError=> b_201CO1Error);
				   
// Drives
FBDiagnosis_101TB1(bWCounter := FALSE,
				   wState := ui101U1State,
				   TimeError :=Time100ms,
				   bError=> b_101U1Error);
FBDiagnosis_101TB2(bWCounter := FALSE,
				   wState := ui101U2State,
				   TimeError :=Time100ms,
				   bError=> b_101U1Error);
FBDiagnosis_101TB3(bWCounter := FALSE,
				   wState := ui101U3State,
				   TimeError :=Time100ms,
				   bError=> b_101U1Error);
FBDiagnosis_101TB4(bWCounter := FALSE,
				   wState := ui101U4State,
				   TimeError :=Time100ms,
				   bError=> b_101U1Error);				   
				   
(*************** PROFINet DIAGNOSIS ************************************)
// 1. AMT
// 0 = No error
// 1 = Profinet device state machine is in boot mode
// 2 = Device not found
// 3 = The stationname is not unique
// 4 = IP could not be set
// 5 = IP conflict
// 6 = DCP set was not successful
// 7 = Watchdog error
// 8 = Datahold error
// 9 = RTC3: Sync mode could not be initiated
// 10 = Profinet controller has a link error
// 11 = The aliasname is not unique
// 12 = The automatic name assignement isn't possible - wrong device type
// 13 = IOC-AR is established but no application ready
// 14 = IOC-AR is established but module difference
// 15 = At least one InputCR is invalid, provider in stop or problemindicator is set
// 16 = At least one OutputCR is invalid, provider in stop or problemindicator is set
// 31 = Only for EtherCAT gateways: WC-State of cyclic EtherCAT frame is 1
b_ProfinetAMTError := (PnIoBoxState <> 0);

END_PROGRAM
